INTERFACE RecipeTableValueType EXTENDS RecipeValue

METHOD ParseAndAssignValues
VAR_INPUT
	rowCount : INT;
END_VAR
END_METHOD

END_INTERFACE

(* stored: Version 1.1.0.1
   Itf RecipeTableValueType: Id {2e1803df-ca34-01f5-379f-db1d47c2c772}
   Method ParseAndAssignValues: Id {b64fcee2-b8ed-0472-2101-b451aab1d8f1} *)
